// TIA Portal V20 export
DATA_BLOCK "DB_MCPManagement"   // DB425
// stored: AutoNumber false, InstanceOfName FB_MCPManagement, InstanceOfType FB
"FB_MCPManagement"
   // VAR
   //    sRT_SingleBlock : R_TRIG;
   //    sSelectionAxe01Jog { S7_SetPoint := 'True'} : Bool;
   //    sSelectionAxe02Jog { S7_SetPoint := 'True'} : Bool;
   //    sSelectionAxe03Jog : Bool;
   //    sSelectionAxe04Jog : Bool;
   //    sSelectionAxe05Jog : Bool;
   //    sSelectionAxe06Jog : Bool;
   //    sSelectionAxe07Jog : Bool;
   //    sSelectionAxe08Jog : Bool;
   //    sSelectionAxe09Jog : Bool;
   //    sSelectionAxe10Jog : Bool;
   //    sSelectionAxe11Jog : Bool;
   //    sSelectionAxe12Jog : Bool;
   //    sSelectionAxe13Jog : Bool;
   //    sSelectionAxe14Jog : Bool;
   //    sSelectionAxe15Jog : Bool;
   //    sSelectionAxe16Jog : Bool;
   //    sSelectionAxe17Jog : Bool;
   //    sResetProgramEnmodeRef : Bool;
   //    sRT_McsWcs { S7_SetPoint := 'True'} : R_TRIG;
   //    sMemoFeedDisable { S7_SetPoint := 'True'} : Bool;
   //    sTONChanRef { S7_SetPoint := 'True'} : TON_TIME;
   //    sFP_TONChanRef { S7_SetPoint := 'True'} : R_TRIG;
   // END_VAR
BEGIN
END_DATA_BLOCK
